// TIA Portal V20 export
DATA_BLOCK "Simulation_DB"   // DB81
// stored: InstanceOfName Unit1.Em7.Simulation, InstanceOfType FB, Namespace Unit1.Em7
"Unit1.Em7.Simulation"
   // VAR_INPUT
   //    simulation { ExternalAccessible := 'False'; ExternalVisible := 'False'; ExternalWritable := 'False'} : Bool;
   // END_VAR
   // VAR
   //    instActuator { ExternalAccessible := 'False'; ExternalVisible := 'False'; ExternalWritable := 'False'} : Array[0..19] of "LER_SimActuator";
   // END_VAR
BEGIN
END_DATA_BLOCK
